// TIA Portal V19 export
DATA_BLOCK "AI"   // DB5
{ S7_Optimized_Access := 'TRUE' }
// stored: MemoryReserve 100
   VAR RETAIN
      Min : Struct
         "LT-1" : Real;
         "LT-2" : Real;
         "CT-1" : Real;
         "CT-2" : Real;
      END_STRUCT;
      Max : Struct
         "LT-1" : Real;
         "LT-2" : Real;
         "CT-1" : Real;
         "CT-2" : Real;
      END_STRUCT;
   END_VAR
   VAR
      PV : Struct
         "LT-1" : Real;
         "LT-2" : Real;
         "CT-1" : Real;
         "CT-2" : Real;
      END_STRUCT;
   END_VAR
   VAR RETAIN
      "LT-1 SET VALVE" : Struct
         LL : Real;
         L : Real;
         H : Real;
         HH : Real;
      END_STRUCT;
   END_VAR
   VAR
      "LT-1" : Struct
         LOW_BUFF : Int;
         HIGH_BUFF : Int;
      END_STRUCT;
   END_VAR
   VAR RETAIN
      "LT-2 SET VALVE" : Struct
         LL : Real;
         L : Real;
         H : Real;
         HH : Real;
      END_STRUCT;
   END_VAR
   VAR
      "LT-2" : Struct
         LOW_BUFF : Int;
         HIGH_BUFF : Int;
      END_STRUCT;
   END_VAR
BEGIN
END_DATA_BLOCK
